(* IEC 61131-3 sources: ATCMcontrol_Engineering/src/TargetBase/Libs/ATCM_ProfibusDP, 8 files *)

(* ---- Profibus_GetEmcyInfo.st ---- *)
(*[[
    UserURL= "ATCMfile:Profibus_GetEmcyInfo.htm"
]]*)
FUNCTION Profibus_GetEmcyInfo:DWORD

VAR_INPUT
   ExecMode:       INT;
END_VAR

VAR_OUTPUT
   ExecStatus:     DWORD;
END_VAR

VAR_INPUT
   Board:          INT;
   NodeId:         INT;
   Timeout:        INT;
END_VAR

VAR_OUTPUT
   StationStatus_1   : BYTE;
   StationStatus_2   : BYTE;
   StationStatus_3   : BYTE;
   MasterAddress     : BYTE;
   IdentNumber       : WORD;
   ExtendedDiagnostic: array[0..99] of BYTE;
END_VAR

inline { STDLIB(PROFI_GET_EMCY_INFO) }

END_FUNCTION

(* ---- Profibus_GetEmcyInfoSlave.st ---- *)
(*[[
    UserURL= "ATCMfile:Profibus_GetEmcyInfoSlave.htm"
]]*)

FUNCTION Profibus_GetEmcyInfoSlave
VAR_INPUT
END_VAR

VAR_INPUT
   ExecMode:       INT;
END_VAR

VAR_OUTPUT
   ExecStatus:     DWORD;
END_VAR

VAR_INPUT
   Board:          INT;
END_VAR

VAR_OUTPUT
   TaskState : WORD;
   ErrorCnt  : WORD;
   LastError : WORD;
   NodeId    : WORD;
END_VAR

inline {STDLIB(PROFI_GET_EMCY_INFO_SLAVE)}

END_FUNCTION

(* ---- Profibus_GetEmcyNode.st ---- *)
(*[[
    UserURL= "ATCMfile:Profibus_GetEmcyNode.htm"
]]*)
FUNCTION Profibus_GetEmcyNode:DWORD

VAR_INPUT
   ExecMode:       INT;
END_VAR

VAR_OUTPUT
   ExecStatus:     DWORD;
END_VAR

VAR_INPUT
   Board:          INT;
END_VAR

VAR_IN_OUT
   NodeId:         INT;
END_VAR

inline {STDLIB(PROFI_GET_EMCY_NODE)}

END_FUNCTION

(* ---- Profibus_GetStatus.st ---- *)
(*[[
    UserURL= "ATCMfile:Profibus_GetStatus.htm"
]]*)
FUNCTION Profibus_GetStatus:DWORD

VAR_INPUT
   ExecMode:       INT;
END_VAR

VAR_OUTPUT
   ExecStatus:     DWORD;
END_VAR

VAR_INPUT
   Board:          INT;
END_VAR

VAR_OUTPUT
   StatusData:     Profibus_StatusType;
END_VAR

inline { STDLIB(PROFI_GET_STATUS) }

END_FUNCTION

(* ---- Profibus_ReadDataRecord.st ---- *)
(*[[
    UserURL= "ATCMfile:Profibus_ReadDataRecord.htm"
]]*)
FUNCTION Profibus_ReadDataRecord : DWORD

VAR_INPUT
   ExecMode		:	INT;
END_VAR

VAR_OUTPUT
   ExecStatus	:	DWORD;
END_VAR

VAR_INPUT
  Board			:	INT;
  RemAddr		:	INT;
  Index			:	INT;
  SlotNumber	:	INT;
  TimeOut		:	INT;
END_VAR

VAR_OUTPUT
  LenDataRead	:	INT;
  DataRead		:	ARRAY [0..255] OF BYTE;
  ErrorCode_1	:	BYTE;
  ErrorCode_2	:	BYTE;
END_VAR

inline { STDLIB(PROFI_READ_DATA_RECORD) }

END_FUNCTION

(* ---- Profibus_ReadDiagnosis.st ---- *)
(*[[
    UserURL= "ATCMfile:Profibus_ReadDiagnosis.htm"
]]*)
FUNCTION Profibus_ReadDiagnosis : DWORD

VAR_INPUT
   ExecMode			:	INT;
END_VAR

VAR_OUTPUT
   ExecStatus		:	DWORD;
END_VAR

VAR_INPUT
  Board				:	INT;
  Timeout			:	INT;
END_VAR

VAR_OUTPUT
  RemAddr			:	INT;
  SlotNumber		:	INT;
  SeqNr				:	INT;
  AlarmType			:	BYTE;
  AlarmSpeckAck		:	BYTE;
  LenDiagUserData	:	INT;
  DiagUserData		:	ARRAY [0..64] OF BYTE;
END_VAR

inline { STDLIB(PROFI_READ_DIAGNOSIS) }

END_FUNCTION

(* ---- Profibus_ReceiveAlarms.st ---- *)
(*[[
    UserURL= "ATCMfile:Profibus_ReceiveAlarms.htm"
]]*)
FUNCTION Profibus_ReceiveAlarms : DWORD

VAR_INPUT
   ExecMode		:	INT;
END_VAR

VAR_OUTPUT
   ExecStatus	:	DWORD;
END_VAR

VAR_INPUT
  Board			:	INT;
  RemAddr		:	INT;
  Index			:	INT;
  SlotNumber	:	INT;
  SeqNr			:	INT;
  Timeout		:	INT;
END_VAR

VAR_OUTPUT
  AlarmType		:	BYTE;
  AlarmSpeckAck	:	BYTE;
END_VAR

inline { STDLIB(PROFI_RECEIVE_ALARMS) }

END_FUNCTION

(* ---- Profibus_WriteDataRecord.st ---- *)
(*[[
    UserURL= "ATCMfile:Profibus_WriteDataRecord.htm"
]]*)
FUNCTION Profibus_WriteDataRecord : DWORD

VAR_INPUT
   ExecMode		:	INT;
END_VAR

VAR_OUTPUT
   ExecStatus	:	DWORD;
END_VAR

VAR_INPUT
  Board			:	INT;
  RemAddr		:	INT;
  Index			:	INT;
  SlotNumber	:	INT;
  Timeout		:	INT;
  LenDataWrite	:	INT;
  DataWrite		:	ARRAY [0..255] OF BYTE;
END_VAR

VAR_OUTPUT
  ErrorCode_1	:	BYTE;
  ErrorCode_2	:	BYTE;
END_VAR

inline { STDLIB(PROFI_WRITE_DATA_RECORD) }

END_FUNCTION
